# EPICS alarm handler configuration: alh_files/mgnt_li26_lgps.alhConfig
GROUP NULL LGPS:LI26:MG01
$ALIAS LGPS
$GUIDANCE
LI26 LGPS magnets
   Group Name: LGPS:LI26:MG01
   Summary PV:  LGPS:LI26:MG01:STATSUMY
$END

GROUP LGPS:LI26:MG01  LGPS:LI26:2
CHANNEL     LGPS:LI26:2           LGPS:LI26:2:STATMSG   -----
   $FORCEPV LGPS:LI26:2:STATMSGSV -DATL 1 0
